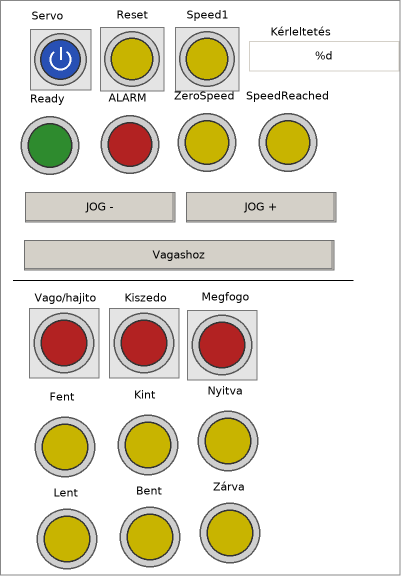
VISUALIZATION TempJozsiNTC  // 401x576
    Lamp1 (16,111 68x69), variable: NTC.bReady, style: Lamp-Lamp1-Green
    Label (13,84 69x30), "Ready"
    Lamp1 (96,110 68x69), variable: NTC.bAlarm, style: Lamp-Lamp1-Red
    Label (93,83 69x30), "ALARM"
    PowerSwitch (19,29 83x61), variable: NTC.bServoON, behaviour: TOGGLE, style: Switch-PowerSwitch-Blue
    Label (13,1 69x30), "Servo"
    PushSwitch (99,27 66x64), variable: NTC.bReset, behaviour: TOGGLE, style: Switch-PushSwitch-Yellow
    Label (98,0 69x30), "Reset"
    Lamp1 (173,108 68x69), variable: NTC.bZeroSpeed, style: Lamp-Lamp1-Yellow
    Label (170,81 69x30), "ZeroSpeed"
    Lamp1 (254,108 68x69), variable: NTC.bSpeedReached, style: Lamp-Lamp1-Yellow
    Label (241,81 93x30), "SpeedReached"
    PushSwitch (174,27 66x64), variable: NTC.bSpeed1, behaviour: TOGGLE, style: Switch-PushSwitch-Yellow
    Label (173,0 69x30), "Speed1"
    Button (186,192 150x30), "JOG +"
        tap NTC.bJogPlus
    Button (25,192 150x30), "JOG -"
        tap NTC.bJogMinus
    Line (13,280) (353,280)
    PushSwitch (29,308 70x70), variable: NTCProcess.bVagoHajlito, behaviour: TOGGLE, style: Switch-PushSwitch-Red
    Label (31,283 69x30), "Vago/hajito"
    PushSwitch (109,308 70x70), variable: NTCProcess.bKiszedo, behaviour: TOGGLE, style: Switch-PushSwitch-Red
    Label (111,283 69x30), "Kiszedo"
    PushSwitch (187,310 70x70), variable: NTCProcess.bMegfogo, behaviour: TOGGLE, style: Switch-PushSwitch-Red
    Label (191,282 69x30), "Megfogo"
    Lamp1 (32,504 70x70), variable: NTCProcess.bVagoHajlitoLent, style: Lamp-Lamp1-Yellow
    Label (11,478 110x30), "Lent"
    Lamp1 (30,412 70x70), variable: NTCProcess.bVagoHajlitoFent, style: Lamp-Lamp1-Yellow
    Label (7,382 110x30), "Fent"
    Lamp1 (115,502 70x70), variable: NTCProcess.bKiszedoBent, style: Lamp-Lamp1-Yellow
    Label (94,476 110x30), "Bent"
    Lamp1 (113,410 70x70), variable: NTCProcess.bKiszedoKint, style: Lamp-Lamp1-Yellow
    Label (90,380 110x30), "Kint"
    Lamp1 (195,498 70x70), variable: NTCProcess.bMegfogoZarva, style: Lamp-Lamp1-Yellow
    Label (174,472 110x30), "Zárva"
    Lamp1 (193,406 70x70), variable: NTCProcess.bMegfogoNyitva, style: Lamp-Lamp1-Yellow
    Label (170,376 110x30), "Nyitva"
    Textfield (249,41 150x30), "%d", text variable: NTC.iDelayFor
        OnMouseClick: write the text variable via VisuDialogs.Numpad, min -10000, max -1
    Label (266,17 69x30), "Kérleltetés"
    Button (24,240 310x30), "Vagashoz"
        OnMouseClick: execute { NTC.bVagashoz:=TRUE; }
END_VISUALIZATION

(* stored: Version 1.1.0.1, ProductVersion 3.1.4024.11
   Visu TempJozsiNTC: Id {abf55278-6971-4570-84e3-983b2bab00c7} *)
